        -0.064878459045791162,136.32800000000003,46.642663706148113,136.32800000000003,-0.064874276850442433,
        136.32800000000003,-9.9999999999999982,136.32800000000003,-5.0116575809989987,136.32800000000006,
        -3.355528608733493,136.328,70.0792111192775,68.082011032644715,70.08246539490186,45.319965612648112,
        70.09379964864479,-14.000000000000004,70.093396079164137,-7.0041486765756957,46.64951683334678,
        68.085052658968351,-10.0,68.09450944594461,-5.0077384299939975,68.094221185452341,-3.34867392142978,
        68.094005674607914,46.655237788220333,45.3255467924812,46.675290764014974,-14.0,46.674585386490143,
        -7.0011083270071328,46.6739994865459,-4.6715366480995613,-10.000000000000004,45.342884475415772,
        -5.0044853711592667,45.342358586139262,-3.3429545257648674,45.341962568857838,-9.9999999999999964,
        -13.999999999999998,-9.9999999999999964,0.0047583223517445906,-9.9999999999999982,-6.9916508524709053,
        -9.9999999999999982,0.0047579065103907177,-10.0,-4.6541980426384946,-4.9931510856853736,-14.000000000000004,
        0.0066625962871976127,-14.0,-3.3229015508666389,-14.0,0.0066621668029032488,-14.000000000000004,
        -4.9935534701073809,-6.991938523768094,-4.9938876273720858,-4.65472309775716,-3.3236053682864015,
        -6.9921553113675454,-3.3241928274392922,-4.6551208717229278,140.32799999999997,136.328,140.32799999999997,
        136.32800000000003,140.32799999999997,136.32800000000003,140.32799999999995,68.077963122328043,
        140.32799999999997,-4.68450785771074,140.32799999999997,-13.999999999999998,140.328,-7.0081868651731956,
        70.075282628673619,136.32800000000003,46.642631530347757,136.32800000000003,-0.06488741702733633,136.328,
        -10.000000000000004,136.32800000000006,-5.011674285092937,136.32800000000006,-3.3555583211233451,136.328,
        -3.3555622946665142,136.32800000000006,-9.9999999999999964,136.32800000000003,-10.0,136.328,
        -5.0116580206210077,136.32800000000003,70.093053791180637,-4.6771185392883865,70.093799613272623,
        -14.000000000000002,70.093396046853826,-7.0041488385579989,-10.0,68.094509232290008,-5.0077386181549555,
        68.094221158296435,46.675291532571208,-14.0,46.675291501195034,-14.000000000000004,46.674585433917038,
        -7.0011081945976974,-10.000000000000002,45.342884578934964,-5.0044853494808894,45.342358591863047,
        -9.9999999999999982,-13.999999999999998,-9.9999999999999964,-14.000000000000002,-9.9999999999999982,
        -4.6541960622305716,-9.9999999999999964,-6.9916498557988653,-9.9999999999999964,-6.99164978602478,
        -9.9999999999999947,-4.6541962631244216,-4.9931503007764517,-14.000000000000002,-4.9931493636029334,
        -13.999999999999998,0.0066635162137103814,-14.000000000000002,-4.9935527110051181,-6.9919384142123366,
        -4.9935532626124521,-6.9919374835265442,-3.3236050032142765,-6.9921542921360684,140.32799999999997,136.328,
        140.32799999999997,-13.999999999999998,140.328,-7.0082015385777172,140.32799999999997,-14.000000000000004,
        140.328,-7.0081991580918,140.32799999999997,-13.999999999999998,140.32799999999997,-7.0082004632995671,
        70.0752640337138,136.32800000000006,-5.01167472585953,136.32800000000003,-10.0,136.32800000000003,
        -5.0116769347395431,136.32800000000003,-10.000000000000002,136.328,70.093790333120168,-14.000000000000002,
        -10.000000000000004,68.094499987629192,-9.9999999999999982,68.094509139194315,-10.0,45.342884545523674,
        -9.9999999999999982,-13.999999999999996,-9.9999999999999947,-14.0,-9.9999999999999947,-6.99164961499385,
        -9.9999999999999982,-6.99164878923034,-4.9931489872730346,-13.999999999999996,-3.3228978875299795,-14.0,
        -4.9935525034925687,-6.9919373739570769,140.32799999999997,136.328,140.32799999999997,-13.999999999999998,
        140.328,-14.000000000000002,140.32799999999997,-14.0,-9.9999999999999947,-14.0,-9.9999999999999982,
        -14.000000000000002,140.32799999999997,136.328];
    Explicit_b_F: ARRAY [0..2499] OF LREAL := [-0.12667340248608433,-0.006063437668709459,-8.3619092552944529E-18,
        -0.0061236585018917839,-0.12667628514510906,-5.4210108624275222E-20,-0.031816478047680653,
        -0.0061304672764802117,-0.12667642439759061,-0.0019406208995937544,-0.056510051660952777,
        -0.0061180833246716549,-0.12667579011109506,-0.0031721409299244907,-8.3619092552944529E-18,
        -0.0061236585018917839,-0.12667628514510906,-5.4210108624275222E-20,-0.031816478047680653,
        -0.0061304672764802117,-0.12667642439759061,-0.0019406208995937544,-0.056510051660952777,
        -0.0061180833246716549,-0.12667579011109506,-0.0031721409299244907,-2.9402207665091273E-17,
        -1.7279472123987727E-19,-3.8997820408061615E-17,-0.0061382781607270242,-2.781635022959441E-17,
        -0.001954554803000661,-4.4508616762898093E-17,-0.0061364362134341171,-3.6496532114819666E-17,
        -0.0031976628134779668,-2.9402207665091273E-17,-1.7279472123987727E-19,-2.781635022959441E-17,
        -0.001954554803000661,-3.6496532114819666E-17,-0.0031976628134779668,-0.031817232753816052,
        1.1705995331054431E-18,-0.12667685008982194,-5.6920614055488983E-19,-0.05651137952441581,
        6.1325185381211345E-19,-0.12667674648668509,2.7105054312137611E-19,-7.7886797082401052E-18,
        1.1655173354219173E-18,-0.031817232753816052,1.1705995331054431E-18,-0.05651137952441581,
        6.1325185381211345E-19,-0.031817266661648996,-0.0019560462806767378,-0.03181709911953777,
        -0.0032004303747762012,-0.031817232753816052,-1.8126505071242027E-19,-0.031817266661648996,
        -0.0019560462806767378,-0.056511442169811681,-0.0019531851178935223,-6.2021869980328007E-18,
        -0.001954554803000661,-0.031817266661648996,-0.0019560462806767387,-0.056511442169811681,
        -0.0019531851178935223,-0.056511148498327293,-0.0031951779041220494,-0.056511379524415789,
        -7.555533889508359E-19,-0.056511442169811694,-0.0019531851178935223,-0.056511148498327293,
        -0.0031951779041220494,2.834532230515472E-17,-0.0031976628134779664,-0.031817099119537742,
        -0.0032004303747762012,-0.056511148498327286,-0.0031951779041220485,-2.9402207665091273E-17,
        -1.7279472123987727E-19,-3.8997820408061615E-17,-0.0061382781607270242,-2.781635022959441E-17,
        -0.001954554803000661,-4.4508616762898093E-17,-0.0061364362134341171,-3.6496532114819666E-17,
        -0.0031976628134779668,-0.031817232753816052,1.1705995331054431E-18,-0.12667685008982194,
        -5.6920614055488983E-19,-0.05651137952441581,6.1325185381211345E-19,-0.12667674648668509,
        2.7105054312137611E-19,-0.031817266661648996,-0.0019560462806767378,-0.03181709911953777,
        -0.0032004303747762012,-0.056511442169811681,-0.0019531851178935223,-0.056511148498327293,
        -0.0031951779041220494,-3.1637633492013779E-17,-2.1218175328720223E-19,-2.9586609384686495E-17,
        -1.2874900798265365E-18,-3.629303244924182E-17,-1.3844753522871539E-18,-3.5260975742571659E-17,
        -0.0019546071360561261,-3.7007716498487636E-17,-0.0032030047769573962,-2.9586609384686495E-17,
        -1.2874900798265365E-18,-3.5260975742571659E-17,-0.0019546071360561261,-0.031819629222642885,
        -5.5904174518783822E-20,-0.056511639234444355,6.7762635780344027E-19,-0.12667689109875555,
        4.87890977618477E-19,1.3640969307162975E-17,4.0657581468206416E-20,-0.031817379490146271,
        2.6427427954334171E-19,-0.056511639234444355,6.7762635780344027E-19,-0.0565116579667842,
        -1.2197274440461925E-19,-9.9828126789839634E-18,-2.1747570920754161E-19,-1.4679504492390652E-17,
        -4.4045713257223618E-20,-0.031819629222642885,-5.5904174518783822E-20,-0.031819495581118705,
        -0.0032010631169945782,-0.031817379490146284,2.6935647722686751E-19,-0.031817277135142374,
        -0.0019560987878057871,-9.8746042199722266E-18,-0.0019574634784031352,-0.031819663167738495,
        -0.0019563921511248318,-0.056511639234444369,-6.6068569885835426E-19,-0.056511591038165096,
        -3.3203691532368573E-19,-0.056511460878431695,-0.0019532373498035932,6.2570323813675166E-18,
        -0.0032030047769573944,-0.031819495581118684,-0.003201063116994579,-3.629303244924182E-17,
        -1.3844753522871539E-18,-5.39196557327058E-17,-1.3755815063409838E-18,-2.2981062650193236E-17,
        -0.0032037800282279736,-3.1515396049813143E-17,-0.0019574634784031361,-3.5260975742571659E-17,
        -0.0019546071360561261,-3.7007716498487636E-17,-0.0032030047769573962,-0.031819629222642885,
        -5.5904174518783822E-20,-0.031817351949048972,2.2700482986415249E-19,-0.12667689109875555,
        4.87890977618477E-19,-0.031819663167738495,-0.0019563921511248322,-0.031817277135142374,
        -0.0019560987878057871,-0.056511460878431688,-0.0019532373498035924,-4.5264312426914288E-17,
        -6.4374503991326826E-20,-1.8829860054818317E-17,-1.4162771898161559E-18,-9.05149995347786E-18,
        -0.0019582276830549272,-4.01097761444595E-17,-1.7999450129153882E-20,-3.2785416075102559E-17,
        -0.0019575161121738087,-4.5264312426914288E-17,-6.4374503991326826E-20,-8.1940908526196947E-18,
        -0.0019579342315898221,-0.031819776023428871,-6.9287295085401768E-19,-0.031819776023428878,
        -6.8609668727598327E-19,-2.6619971612698751E-17,3.5575383784680614E-19,-0.031819786518259209,
        8.7752613335545515E-19,-1.8776920495614923E-17,-1.4095957935146237E-18,-0.031819748476883458,
        -1.1892342579450377E-18,-1.1073949933725112E-17,-0.0019575161121738074,1.2611473551669278E-17,
        -0.0019582276830549259,7.93648695753598E-18,-0.0032044132383236136,-3.4094373146186072E-17,
        -1.3349239248727773E-18,-4.5264312426914288E-17,-6.4374503991326826E-20,-9.0567409698389962E-18,
        -0.001958227683054928,-5.43860797190673E-17,-0.0019575161121738087,-0.031817389976958411,
        -1.5280474368467578E-18,-0.0565116579667842,-1.2197274440461925E-19,-0.031819673649245137,
        -0.0019564446946577791,-4.0445883408782404E-17,-2.0629487430378485E-18,-1.4750814078637623E-17,
        -8.2818133307315491E-19,-4.0447185391066563E-17,6.3866284222974246E-19,-4.8277910069457279E-17,
        -9.9229909770841285E-19,-2.6619429395807223E-17,-9.9568722949743E-19,-4.0445883408782404E-17,
        -2.0629487430378485E-18,-4.3236735011029394E-17,-1.334067109051033E-18,-0.010939895258464375,
        -0.12940337663776541,1.8973538018496328E-19,-0.12940857748967641,-0.011001415774033131,
        -1.1907589172500954E-17,-0.0034622111951241163,-0.12940866066139117,-0.011010925708052186,
        -0.032495995972325727,-0.005684687311205988,-0.12940746957634541,-0.010999089451642668,-0.0577221130716327,
        1.8973538018496328E-19,-0.12940857748967641,-0.011001415774033131,-1.1907589172500954E-17,
        -0.0034622111951241163,-0.12940866066139117,-0.011010925708052186,-0.032495995972325727,
        -0.0056846873112059888,-0.12940746957634541,-0.010999089451642668,-0.057722113071632712,
        -1.8499199568033919E-18,-3.1316290367649179E-17,-2.5207700510287978E-18,-0.12940951062758926,
        -3.3627208005995723E-18,-0.032497207130407976,-2.3445871979999033E-18,-0.12940931580424303,
        -1.5958100726271018E-18,-0.057724329102651205,-1.8499199568033919E-18,-3.1316290367649179E-17,
        -3.3627208005995723E-18,-0.032497207130407976,-1.5856456772600502E-18,-0.057724329102651212,
        -0.0034781423641150754,-1.4472616695023789E-17,-0.011018053990055782,-1.9238659330986924E-17,
        -0.0057127737954156535,4.3457025358881879E-18,-0.011016492215632667,-1.3649088912055796E-17,
        -5.1838416371963181E-19,1.1910130271342717E-17,-0.0034781423641150754,-1.4472616695023789E-17,
        -0.0057127737954156543,4.3465495688354422E-18,-0.0034805192947300781,-0.032497220518183073,
        -0.0034774059198201877,-0.057724356242492864,-0.0034781423641150754,7.140911261827379E-18,
        -0.0034805192947300781,-0.032497220518183073,-0.00571704223028016,-0.032496943931058939,
        -6.7593229190893167E-19,-0.032497207130407955,-0.0034805192947300781,-0.032497220518183059,
        -0.0057170422302801607,-0.032496943931058939,-0.0057115870095412712,-0.057723849103550343,
        -0.0057127737954156535,4.3457025358881879E-18,-0.0057170422302801616,-0.032496943931058932,
        -0.0057115870095412712,-0.05772384910355035,3.7980957354882827E-18,-0.057724329102651191,
        -0.0034774059198201864,-0.057724356242492864,-0.00571158700954127,-0.057723849103550329,
        -1.8499199568033919E-18,-3.1316290367649179E-17,-2.5207700510287978E-18,-0.12940951062758926,
        -3.3627208005995723E-18,-0.032497207130407976,-2.3445871979999033E-18,-0.12940931580424303,
        -1.5856456772600502E-18,-0.057724329102651212,-0.0034781423641150754,-1.4472616695023789E-17,
        -0.011018053990055782,-1.9238659330986924E-17,-0.0057127737954156543,4.3465495688354422E-18,
        -0.011016492215632667,7.9917558573443237E-18,-0.0034805192947300781,-0.032497220518183073,
        -0.0034774059198201877,-0.057724356242492864,-0.0057170422302801607,-0.032496943931058939,
        -0.005711587009541272,-0.05772384910355035,-1.1180834903756764E-18,-2.8703842234969904E-17,
        -2.2514135738019303E-18,-1.6261338521388058E-17,-2.1785687403380605E-18,-3.0005983337805979E-17,
        -2.4496192834594366E-18,-0.032499690181368147,-2.4530074152484538E-18,-0.057724640166312291,
        -2.2514135738019303E-18,-1.6261338521388058E-17,-2.447925217564928E-18,-0.032499690181368147,
        -0.0034782384082034431,-2.9130521847259457E-18,-0.0057203209764982678,-1.5056010637445189E-17,
        -0.011020049672395411,1.9245435594564958E-17,1.7885100681274552E-18,5.3299548205976849E-18,
        -0.0034823937966747143,-4.7944182396961535E-18,-0.0057203209764982686,-1.5054740088024307E-17,
        -0.0057212109064913585,-3.6574882662440689E-17,2.1345230270808369E-19,1.4522843101818009E-17,
        -8.3348042009823153E-19,-8.3925083205140145E-18,-0.0034782384082034418,-2.9136874594363864E-18,
        -0.0034775019361867527,-0.057724381593873116,-0.0034823937966747156,1.6840391419954779E-17,
        -0.003481014589598143,-0.032499703597191981,3.1001405869507392E-19,-0.03249737675610765,
        -0.0034806155086637754,-0.032497234404046518,-0.0057203209764982695,-1.499333019934837E-17,
        -0.0057195819017150417,7.3615633445871242E-18,-0.0057179316027686257,-0.032499426937493366,
        2.9341221292888964E-18,-0.057724640166312263,-0.0034775019361867514,-0.057724381593873109,
        -2.1751806085490433E-18,-3.0005401002654742E-17,-2.1590869825512116E-18,-1.8180291663392675E-17,
        -2.6393546636444E-18,-0.057724722338242183,-1.0333801956502464E-18,-0.032497376756107664,
        -2.447925217564928E-18,-0.032499690181368147,-2.4496192834594366E-18,-0.057724640166312291,
        -0.0034782384082034418,-2.9136874594363864E-18,-0.0034819660630087974,-1.42590585131973E-17,
        -0.011020049672395411,-2.3488223627361748E-18,-0.0034806155086637754,-0.032497234404046539,
        -0.003481014589598143,-0.032499703597191981,-0.0057179316027686248,-0.032499426937493379,
        -2.4321715627988556E-19,-2.4769572718320691E-17,-3.2932640989247197E-18,-4.3098028973033865E-17,
        -3.0493186101154812E-20,-0.032497435184955785,-1.1608586542120186E-18,-7.0482140936622365E-18,
        -1.7508171019746388E-18,-0.032499859870392257,-2.3045448321122832E-19,-4.6363830675621824E-17,
        -1.2468324983583301E-18,-0.032499904406537286,-0.0034824901317153855,-1.3784825941853297E-17,
        -0.0034824901317153868,-3.5417518019136094E-17,2.2535452699392677E-19,-1.0840645296315756E-17,
        -0.0034829857776749878,-6.0625324408542479E-18,-5.8614679949997583E-19,-4.309872711347086E-17,
        -0.0034820623747332268,-5.69567188348657E-17,9.4867690092481638E-19,-0.032499859870392236,
        2.6495190590114515E-18,-0.032497435184955743,2.8426425709854319E-18,-0.05772474772329142,
        -1.74022919013396E-18,-3.8454607591075591E-17,-2.3045448321122832E-19,-4.6363830675621824E-17,
        -4.072534410398676E-18,-0.0324974351849558,-3.0823528950583989E-18,-0.032499859870392278,
        -0.0034828894057362539,-1.4940390640144977E-17,-0.0057212109064913577,-1.4962837013247215E-17,
        -0.0034811108404072628,-0.032499717489793044,-4.6570117914014579E-19,-5.4131969834891012E-17,
        -7.75458663211312E-19,-5.4659205244755268E-17,-4.7875783090603467E-19,-1.0848096539273634E-17,
        -1.1109398035093036E-18,-5.4060977885999261E-17,-2.4568260686969107E-18,-5.4074900990069754E-17,
        8.7612459859210622E-19,-3.2500058616106466E-17,-2.7055760048624738E-18,-2.1687985305904772E-17,
        -0.021835439137868347,-0.0011520122606157824,8.3760970571609625E-19,-0.0011623928796879576,
        -0.021835986823640203,2.9815559743351372E-19,-0.0046660193730712375,-0.0011641448432321742,
        -0.021836028047420925,-0.00034855849507587592,-0.0088399634659200779,-0.0011621335886920921,
        -0.021835908054478017,-0.00058417725377516751,8.3760970571609625E-19,-0.0011623928796879576,
        -0.021835986823640203,2.9815559743351372E-19,-0.0046660193730712375,-0.0011641448432321742,
        -0.021836028047420925,-0.00034855849507587592,-0.0088399634659200761,-0.0011621335886920921,
        -0.021835908054478017,-0.00058417725377516751,-1.1794933790516132E-19,3.5151867311053464E-19,
        -1.6721489169983957E-18,-0.0011652903420256554,-2.9172079401234121E-18,-0.00035096037140803615,
        -2.1520989607363636E-18,-0.0011650045622868016,-2.9730327053033908E-18,-0.00058857662244823472,
        -1.1794933790516132E-19,3.5151867311053464E-19,-2.9172079401234121E-18,-0.00035096037140803615,
        -2.9730327053033908E-18,-0.00058857662244823472,-0.0046661626879632477,3.7269449679189215E-19,
        -0.021836104506786864,2.2869889575866109E-19,-0.0088402156943794986,4.7137383514701814E-19,
        -0.021836084179334414,3.1340219048409113E-19,-2.8197197418503624E-18,3.5278922253141609E-19,
        -0.0046661626879632477,3.7269449679189215E-19,-0.0088402156943794968,4.6925625277888239E-19,
        -0.0046661729227340945,-0.00035135054557220417,-0.00466614122182821,-0.00058929774581286808,
        -0.0046661626879632477,3.7269449679189215E-19,-0.0046661729227340945,-0.00035135054557220417,
        -0.0088402343122757146,-0.00035088561017350455,-2.1543753617821095E-19,-0.00035096037140803615,
        -0.0046661729227340919,-0.000351350545572204,-0.0088402343122757129,-0.00035088561017350455,
        -0.0088401787462571157,-0.00058844410776131336,-0.0088402156943794986,3.0239076216978522E-19,
        -0.00884023431227572,-0.00035088561017350455,-0.0088401787462571157,-0.00058844410776131336,
        2.430455163027808E-18,-0.00058857662244823472,-0.0046661412218282064,-0.00058929774581286819,
        -0.00884017874625711,-0.00058844410776131336,-1.1794933790516132E-19,3.5151867311053464E-19,
        -1.6721489169983957E-18,-0.0011652903420256554,-2.9172079401234121E-18,-0.00035096037140803615,
        5.4284224007159973E-19,-0.0011650045622868016,-2.9730327053033908E-18,-0.00058857662244823472,
        -0.0046661626879632477,3.7269449679189215E-19,-0.021836104506786864,2.2869889575866109E-19,
        -0.0088402156943794968,4.6925625277888239E-19,-0.021836084179334414,3.1340219048409113E-19,
        -0.0046661729227340945,-0.00035135054557220417,-0.00466614122182821,-0.00058929774581286808,
        -0.0088402343122757129,-0.00035088561017350455,-0.0088401787462571123,-0.00058844410776131336,
        -1.3346592270767604E-18,2.82326669231699E-19,-1.99168547890518E-19,2.2658131339052534E-19,
        -1.578684125224804E-18,2.3727510434961088E-19,-8.3673620298924025E-19,-0.00035097205163314076,
        3.0059081715686983E-19,-0.00058966848483959448,-1.99168547890518E-19,2.2658131339052534E-19,
        -8.3673620298924025E-19,-0.00035097205163314076,-0.004666697129121284,4.8174998875088332E-19,
        -0.008840269714523688,4.3410438546782892E-19,-0.021836113712710516,2.0837010502455788E-19,
        7.9059491036817479E-18,3.9048218868423246E-19,-0.0046661931893067525,4.5655075857006788E-19,
        -0.0088402697145236846,4.3198680309969317E-19,-0.0088402739021540347,5.6158284402960112E-19,
        1.3670317675296357E-18,4.4993331366964366E-19,-1.5821516663526262E-18,4.0562290261640307E-19,
        -0.0046666971291212866,4.8302053817176477E-19,-0.0046666756618988928,-0.00058943885502096274,
        -0.0046661931893067577,2.9116757561866574E-19,-0.0046661752611696682,-0.00035136226893268138,
        -1.4712035851521137E-18,-0.0003515548854198116,-0.004666707372365379,-0.00035142767883477574,
        -0.008840269714523688,9.6561755986990239E-20,-0.0088402602471837673,2.9730856448625942E-19,
        -0.0088402384954132315,-0.00035089728892171812,3.0045846825886135E-19,-0.00058966848483959437,
        -0.0046666756618988928,-0.00058943885502096285,-1.5888485205918556E-18,2.3611043404713622E-19,
        -6.3560558268574647E-19,3.1890790464124408E-19,-1.3013867141174274E-18,-0.00058978898971890226,
        -1.4744726029329233E-18,-0.00035155488541981176,-8.3673620298924025E-19,-0.00035097205163314076,
        2.9381455357883543E-19,-0.00058966848483959448,-0.0046666971291212866,4.8302053817176477E-19,
        -0.004666187775523677,4.7222086809427244E-19,-0.021836113712710516,2.0837010502455788E-19,
        -0.0046667073723653842,-0.00035142767883477574,-0.0046661752611696682,-0.00035136226893268138,
        -0.0088402384954132263,-0.00035089728892171796,-1.8489761437244689E-18,1.232432938255007E-19,
        -1.4251329337553603E-19,1.5386230185264307E-19,-2.7136156303169605E-18,-0.00035169687999964154,
        -4.9415935230040384E-19,4.258458142320995E-19,5.2317519382753894E-19,-0.00035156662712727745,
        -1.8489761437244689E-18,1.232432938255007E-19,-2.4459399840948007E-19,-0.00035163144666093126,
        -0.0046667276446882341,4.1102273765514924E-19,-0.0046667276446882315,4.0890515528701349E-19,
        -9.5356553834500477E-19,4.2679872629776058E-19,-0.00466672998743669,5.14784273693801E-19,
        -1.4592789494415493E-19,3.2237967214500863E-19,-0.0046667222297373193,1.0630263488041469E-19,
        5.2647068138795021E-19,-0.00035156662712727729,2.6900972311408528E-18,-0.00035169687999964138,
        -5.7968817327716179E-20,-0.00058993018680938666,1.5512217288880434E-18,2.3791037906005161E-19,
        -1.8489761437244689E-18,1.232432938255007E-19,-1.6953893834886855E-20,-0.00035169687999964171,
        -4.890516774540114E-18,-0.00035156662712727745,-0.0046661955302668917,3.2441361879839703E-19,
        -0.0088402739021540312,5.5946526166146537E-19,-0.00466670971258821,-0.00035143941031378837,
        -2.460318683737051E-18,2.4156320864508578E-19,-1.9600474748362518E-18,2.4520144624712663E-19,
        -2.4653401353443424E-18,2.413514504082722E-19,-9.535282635186516E-19,2.5770977420212088E-19,
        -9.47597120032705E-19,2.5845092803096839E-19,-2.460318683737051E-18,2.4156320864508578E-19,
        -2.7015815614391379E-18,1.7057475020245581E-19,-0.0034982247754591846,-0.037913871321265488,
        3.2864878353466853E-19,-0.03791553438554341,-0.003516249659905755,6.0562855728682474E-20,
        -0.0010483412940467669,-0.037915602504622059,-0.00352001142228519,-0.0081901839499625134,
        -0.0017637665131279233,-0.037915222177636647,-0.003516769828667967,-0.015456721801501918,
        3.2864878353466853E-19,-0.03791553438554341,-0.003516249659905755,6.0562855728682474E-20,
        -0.0010483412940467669,-0.037915602504622059,-0.00352001142228519,-0.0081901839499625134,
        -0.0017637665131279229,-0.037915222177636647,-0.003516769828667967,-0.015456721801501924,
        -2.0159384144652348E-19,-1.1845226371759356E-18,-4.7433845046240819E-20,-0.037915859870396064,
        -9.1564261598189867E-19,-0.0081905711372341986,-4.8111471404044259E-19,-0.037915794999810175,
        -3.7438856268640075E-19,-0.015457430339336756,-2.0159384144652348E-19,-1.1845226371759356E-18,
        -9.1564261598189867E-19,-0.0081905711372341986,-3.6930636500287495E-19,-0.015457430339336761,
        -0.0010530089868256581,5.6347808024908262E-18,-0.0035218080110374283,-2.732951804316E-18,
        -0.0017719955998451308,3.356897449087199E-18,-0.0035214299089605374,8.1734444245303711E-18,
        -2.0413494028828638E-19,4.2188593520368564E-18,-0.0010530089868256581,5.6347808024908262E-18,
        -0.0017719955998451308,3.356897449087199E-18,-0.0010539568187064221,-0.0081905849637701356,
        -0.0010531016854318472,-0.015457456534433,-0.0010530089868256581,5.6347808024908262E-18,
        -0.0010539568187064221,-0.0081905849637701356,-0.0017736905237788257,-0.0081904966580441437,
        4.3113977015243887E-19,-0.0081905711372341934,-0.0010539568187064217,-0.00819058496377013,
        -0.0017736905237788255,-0.0081904966580441437,-0.0017721939819592,-0.015457294593549919,
        -0.0017719955998451308,-2.0464316005663896E-18,-0.0017736905237788266,-0.0081904966580441437,
        -0.0017721939819592,-0.015457294593549924,9.7493492228969969E-19,-0.015457430339336754,
        -0.0010531016854318466,-0.015457456534433001,-0.0017721939819591993,-0.015457294593549914,
        -2.0159384144652348E-19,-1.1845226371759356E-18,-4.7433845046240819E-20,-0.037915859870396064,
        -9.1564261598189867E-19,-0.0081905711372341986,-4.8450284582945979E-19,-0.037915794999810175,
        -3.6930636500287495E-19,-0.015457430339336761,-0.0010530089868256581,5.6347808024908262E-18,
        -0.0035218080110374283,-2.732951804316E-18,-0.0017719955998451308,3.356897449087199E-18,
        -0.0035214299089605374,8.18699695168644E-18,-0.0010539568187064221,-0.0081905849637701356,
        -0.0010531016854318472,-0.015457456534433004,-0.0017736905237788255,-0.0081904966580441437,
        -0.0017721939819591997,-0.015457294593549924,-4.7010328572613669E-19,-1.3141914699997482E-19,
        -8.4385657370209671E-20,-1.1857402470376137E-18,-8.6736173798840355E-19,-3.407203265220224E-18,
        -5.8720559068404371E-19,-0.0081914952946237352,-2.388632911257127E-19,-0.015457540044886605,
        -8.4385657370209671E-20,-1.1857402470376137E-18,-5.9038196423624734E-19,-0.0081914952946237282,
        -0.001053044746302335,1.5328649367342666E-18,-0.0017745168956370212,2.7445985073407467E-18,
        -0.0035225506987666363,7.3653749928497686E-18,1.262820245237755E-18,9.6305528520445813E-18,
        -0.0010544292673404124,7.4725246606774376E-18,-0.001774516895637021,2.7442808699855263E-18,
        -0.0017748480792266457,-1.0456621733854338E-18,-4.70950318673391E-19,5.2720720300536742E-18,
        -1.9566461081574338E-19,1.9956890330699367E-18,-0.0010530447463023354,1.5330766949710802E-18,
        -0.0010531374576252502,-0.015457465979431909,-0.0010544292673404132,2.0594017925712211E-18,
        -0.001054141160788231,-0.0081915091323479083,3.2314306937751558E-19,-0.00819063094036294,
        -0.0010539926448452485,-0.0081905901342984883,-0.0017745168956370219,-8.0768826685433809E-18,
        -0.001774334854501361,-4.3972656665522934E-18,-0.001774021536753176,-0.0081914208010279415,
        4.2775163836342167E-19,-0.015457540044886595,-0.0010531374576252493,-0.015457465979431904,
        -8.6820877093565785E-19,-3.4073620838978341E-18,-3.4050724479622874E-19,-2.993361496037494E-18,
        -2.447925217564928E-19,-0.015457567403298908,-3.4813054132151744E-19,-0.0081906309403629463,
        -5.9038196423624734E-19,-0.0081914952946237282,-2.405573570202213E-19,-0.015457540044886605,
        -0.0010530447463023354,1.5330766949710802E-18,-0.0010543228028200187,5.2656332561655615E-18,
        -0.0035225506987666363,7.3810451023739732E-18,-0.0010539926448452492,-0.0081905901342984935,
        -0.001054141160788231,-0.0081915091323479083,-0.0017740215367531753,-0.0081914208010279415,
        -4.6609629359195911E-19,-4.648622693650007E-19,-2.7782680669941051E-19,3.4962161709370553E-18,
        -1.7575933655526732E-19,-0.00819065093434982,-3.6348301349050163E-19,1.1533177448757402E-17,
        8.9573734172142261E-20,-0.00819155512097787,-4.6485265339037978E-19,-4.55227269589983E-19,
        -6.9393174203808555E-19,-0.0081915699426062215,-0.0010544651240993646,-2.1534753892756518E-18,
        -0.0010544651240993646,-2.1535812683940586E-18,-1.4930700529461648E-20,-2.1646721060471696E-18,
        -0.0010546495763118805,4.4861511864547916E-18,4.0064658405128406E-19,-1.907404046292152E-18,
        -0.0010543586543143618,-2.3973149989664835E-18,8.1950437646853558E-20,-0.00819155512097786,
        4.921261423547485E-19,-0.0081906509343498083,3.5998900258307764E-19,-0.015457576859199004,
        -4.6120943977996653E-19,1.749573022333359E-18,-4.6485265339037978E-19,-4.55227269589983E-19,
        -8.4745646372792749E-19,-0.0081906509343498256,8.8726701224887961E-20,-0.00819155512097787,
        -0.001054613705821476,-5.1583777092194857E-18,-0.0017748480792266462,-1.0256510200065509E-18,
        -0.0010541770006516429,-0.0081915143053841559,4.1312398320618707E-20,-3.1012490089715603E-18,
        -1.0894961284058438E-18,5.3833863454703946E-18,4.23171206500766E-20,7.7514036411160156E-18,
        -1.3193265813930833E-20,-2.1547194689169316E-18,-1.1759897521695683E-20,-7.5663467944756522E-18,
        4.5249235199094131E-20,-8.4940530125110242E-18,5.4294849001241571E-22,-5.4233692790932017E-18,
        -0.90852126123084109,-0.043908146081154252,1.1237416704633352E-16,-0.044340059223466725,
        -0.90854213589311628,5.4210108624275222E-18,-0.22499743169378195,-0.044391150716473024,-0.90854320277576739,
        -0.013973130057841329,-0.40175302414947389,-0.044302834795567785,-0.90853861186181406,-0.02289738328452481,
        1.1237416704633352E-16,-0.044340059223466725,-0.90854213589311628,5.4210108624275222E-18,
        -0.22499743169378195,-0.044391150716473024,-0.90854320277576739,-0.013973130057841329,-0.40175302414947389,
        -0.044302834795567785,-0.90853861186181406,-0.02289738328452481,-2.0211137857729586E-16,
        -3.3610267347050637E-18,1.4233541645661263E-17,-0.044446387153773116,-1.2255042087464668E-16,
        -0.014073066200566241,-1.7068052700353054E-16,-0.044433312973263257,-1.4178653910679184E-16,
        -0.02308043023166,-2.0211137857729586E-16,-3.3610267347050637E-18,-1.2254660922638404E-16,
        -0.014073066200566246,-1.4178653910679184E-16,-0.02308043023166,-0.22500289657472694,1.6127507315721878E-18,
        -0.90854626790451765,5.4210108624275222E-19,-0.4017626395980568,1.0543866127421531E-17,-0.90854551524313676,
        7.48099499014998E-18,-2.9203154922486513E-17,7.37257477290143E-18,-0.22500289657472694,
        1.6127507315721878E-18,-0.40176263959805669,1.0489656018797255E-17,-0.2250031571391346,
        -0.014084282907403574,-0.22500194445913865,-0.023101232532859166,-0.22500289657472694,
        1.7821573210230479E-17,-0.2250031571391346,-0.014084282907403586,-0.40176311984350016,-0.014063877541696803,
        -1.2255465603938295E-16,-0.014073066200566236,-0.2250031571391346,-0.014084282907403574,
        -0.40176311984350005,-0.014063877541696803,-0.4017609942320583,-0.023063772260979193,-0.40176263959805669,
        5.0957502106818708E-18,-0.40176311984350022,-0.014063877541696813,-0.4017609942320583,-0.023063772260979193,
        2.0403837853229939E-16,-0.02308043023166,-0.22500194445913849,-0.023101232532859169,-0.401760994232058,
        -0.023063772260979186,-2.0211137857729586E-16,-3.3610267347050637E-18,1.4233541645661263E-17,
        -0.044446387153773116,-1.2254660922638404E-16,-0.014073066200566246,1.9888333601530972E-18,
        -0.044433312973263257,-1.4178653910679184E-16,-0.02308043023166,-0.22500289657472694,1.6127507315721878E-18,
        -0.90854626790451765,5.9631119486702744E-18,-0.40176263959805669,1.0489656018797255E-17,
        -0.90854551524313676,7.48099499014998E-18,-0.2250031571391346,-0.014084282907403586,-0.22500194445913865,
        -0.023101232532859166,-0.40176311984350005,-0.014063877541696808,-0.40176099423205819,-0.023063772260979193,
        -1.1948500863853337E-16,-7.8316666303132609E-18,-1.0077230382823216E-16,-2.5478751053409354E-18,
        -4.0905762121751926E-17,1.6703489719854803E-18,-8.65074749030817E-18,-0.014073452133259199,
        -5.3407121390278145E-17,-0.023119416718676764,-1.0077092739969287E-16,-2.5343225781848666E-18,
        -8.643971226730135E-18,-0.014073452133259209,-0.22502056771591866,8.2263839837337649E-18,
        -0.40176453880416918,6.5323180892251642E-18,-0.90854657053851451,5.5294310796760726E-18,
        2.45051555019675E-16,2.6834003769016235E-18,-0.22500396954755839,9.4867690092481638E-19,
        -0.40176453880416907,6.478107980600889E-18,-0.40176467697335466,-2.439454888092385E-19,
        5.3732382042023796E-17,8.3331101350878067E-18,-4.1341984089587891E-17,7.0235971986326584E-18,
        -0.22502056771591855,8.1518450843753865E-18,-0.22501961554900995,-0.023105898263657981,-0.22500396954755847,
        1.1858461261560205E-17,-0.225003234379625,-0.014084670139843564,-5.3978445113201171E-17,
        -0.014094294168846267,-0.22502082855573682,-0.014086833295573026,-0.40176453880416929,
        6.6407383064737147E-18,-0.40176418862008356,6.3967928176644762E-18,-0.40176325784096573,
        -0.014064262811759857,1.1939607017907167E-16,-0.023119416718676764,-0.22501961554900987,
        -0.023105898263657981,-4.1339442990746128E-17,1.6195269951502222E-18,-4.3272795692854069E-18,
        2.1819568721270777E-18,-8.3520836731063031E-17,-0.023124920378727248,-5.4079242033924432E-17,
        -0.014094294168846278,-8.643971226730135E-18,-0.014073452133259209,-2.2653726767726812E-16,
        -0.023119416718676764,-0.22502056771591855,8.1518450843753865E-18,-0.22500376942411082,
        4.2283884726934673E-18,-0.90854657053851451,1.0950441942103595E-17,-0.225020828555737,-0.014086833295573026,
        -0.225003234379625,-0.014084670139843564,-0.4017632578409655,-0.014064262811759858,-6.8140584528386856E-17,
        -4.7298319774680131E-18,-1.5717712775840248E-16,-4.8427867988345792E-18,-1.8241786255363338E-16,
        -0.014099813725742058,-9.7153620258884181E-18,1.44774871344705E-17,-1.9124479289697044E-16,
        -0.014094682296279696,-6.8139128690508763E-17,-4.7162794503119443E-18,-6.6146920433456449E-17,
        -0.014097649905087963,-0.22502164116342194,6.8711312681268844E-18,-0.2250216411634221,
        1.5517643593698782E-18,-1.0201159574812646E-16,2.2158381900172497E-18,-0.22502171855946634,
        2.1480755542369057E-18,1.5798011499239956E-17,4.91865166871488E-19,-0.22502144099999252,
        2.6766241133235891E-18,-1.8120999357084874E-17,-0.014094682296279686,-9.6193296654934618E-18,
        -0.014099813725742047,1.9217822320484468E-16,-0.023129589494450122,-1.5185585502551415E-16,
        -3.1611269591530489E-18,-6.8139128690508763E-17,-4.7162794503119443E-18,-9.698950762535366E-18,
        -0.014099813725742063,-1.9135406014716624E-16,-0.014094682296279696,-0.22500404688447739,
        8.40256683676266E-18,-0.40176467697335472,1.0625181290357943E-17,-0.22502090585531667,-0.0140872207964491,
        -2.8013481348918148E-16,5.2482161411876449E-18,-1.0580415599095554E-16,-2.786738913454531E-18,
        -1.0705883760614638E-16,1.0608240631412857E-17,-1.0176638301861879E-16,2.2463313761184045E-18,
        -1.0165657313794115E-16,-3.1509625637859973E-18,-2.8013342961601668E-16,5.2583805365546965E-18,
        -5.7474348667278365E-20,-2.9607205860406696E-20,-0.077953938048960669,-0.91495630205656719,
        1.5395670849294163E-17,-0.91499336154188149,-0.078388923478923359,-1.2000762796698927E-17,
        -0.024548090137893282,-0.91499404071464974,-0.0784581439271197,-0.22706440144138565,-0.040393877243513461,
        -0.91498555513722191,-0.07837495020825766,-0.405131234178429,1.5395670849294163E-17,-0.91499336154188149,
        -0.078388923478923359,-1.2000762796698927E-17,-0.024548090137893282,-0.91499404071464974,
        -0.0784581439271197,-0.22706440144138565,-0.040393877243513461,-0.91498555513722191,-0.07837495020825766,
        -0.405131234178429,-1.2197274440461925E-18,-6.8118389618190833E-17,-4.9873299934333204E-18,
        -0.91500006722362592,-4.8382521947165635E-18,-0.22707303152550876,-3.2526065174565133E-18,
        -0.91499867394199985,-9.7849246066816775E-18,-0.4051470246964986,-1.2197274440461925E-18,
        -6.8118389618190833E-17,-4.8382521947165635E-18,-0.22707303152550876,-9.7849246066816775E-18,
        -0.4051470246964986,-0.024660732712307117,1.417594340524797E-17,-0.078507952497007219,
        1.9447876468958736E-17,-0.040592464909515784,1.8488357546309064E-16,-0.078497094095205028,
        7.5948362182609586E-17,-1.3823577699190182E-18,2.7769805769142786E-16,-0.024660732712307103,
        1.4168320108722682E-17,-0.040592464909515784,1.8488357546309064E-16,-0.024678049245177087,
        -0.22707314681162666,-0.02465616095779212,-0.405147254584257,-0.024660732712307117,1.8708416706005732E-16,
        -0.024678049245177087,-0.22707314681162666,-0.0406235469714099,-0.22707117636130061,5.9089018400459992E-18,
        -0.22707303152550867,-0.024678049245177074,-0.22707314681162657,-0.0406235469714099,-0.22707117636130061,
        -0.040585198407018679,-0.405143641589301,-0.040592464909515784,1.1975351808281298E-17,-0.040623546971409907,
        -0.2270711763613007,-0.040585198407018679,-0.405143641589301,1.1763593571467723E-17,-0.40514702469649849,
        -0.0246561609577921,-0.405147254584257,-0.040585198407018672,-0.405143641589301,-1.2197274440461925E-18,
        -6.8118389618190833E-17,-4.9873299934333204E-18,-0.91500006722362592,-4.8382521947165635E-18,
        -0.22707303152550876,-3.2526065174565133E-18,-0.91499867394199985,-9.7849246066816775E-18,
        -0.4051470246964986,-0.024660732712307103,1.4168320108722682E-17,-0.078507952497007219,
        1.9447876468958736E-17,-0.040592464909515784,1.8488357546309064E-16,-0.078497094095205028,
        7.5948362182609586E-17,-0.024678049245177087,-0.22707314681162666,-0.024656160957792109,-0.405147254584257,
        -0.0406235469714099,-0.22707117636130061,-0.040585198407018679,-0.405143641589301,-1.4094628242311558E-18,
        6.5815518792843204E-18,-1.4894227344519617E-17,-4.6953577365147631E-17,7.3183646642771549E-19,
        -1.4633468251707381E-16,5.2922618544448685E-18,-0.22709100233229687,-9.5680841721845766E-18,
        -0.40514926269585039,-1.4894227344519617E-17,-4.6953577365147631E-17,5.2922618544448685E-18,
        -0.22709100233229687,-0.02466142784965503,1.1036924006018259E-16,-0.040646457087583146,
        1.5888644024596166E-17,-0.0785223958657716,8.3937576941112146E-17,2.8192644616412132E-17,
        2.9900517147960978E-16,-0.02469114725936063,9.6381337969225073E-17,-0.040646457087583146,
        1.5888644024596166E-17,-0.040652897782438434,1.9426361832098477E-16,-1.5178830414797062E-18,
        1.7948585800671261E-16,6.5052130349130266E-19,2.657311762126191E-17,-0.02466142784965503,
        1.1037008709312984E-16,-0.024656855942051376,-0.40514743808224646,-0.024691147259360651,
        9.639658456227565E-17,-0.024681633887332338,-0.22709111782296573,7.15573433840433E-18,-0.22707425188322058,
        -0.024678745617735788,-0.22707324731405812,-0.040646457087583153,1.5893726222279692E-17,
        -0.040641311777483369,4.953956895311501E-17,-0.04062998370810441,-0.22708914685042259,
        1.0299920638612292E-18,-0.40514926269585017,-0.024656855942051355,-0.40514743808224646,
        7.3183646642771549E-19,-1.4633468251707381E-16,-2.0464316005663896E-18,-2.880081427254072E-17,
        6.2341624917916505E-18,-0.40514985034555978,7.26415455565288E-18,-0.22707425188322075,
        5.2922618544448685E-18,-0.22709100233229687,-9.5680841721845766E-18,-0.40514926269585039,
        -0.02466142784965503,1.1037008709312984E-16,-0.02468816702271235,1.2348385118252092E-16,-0.0785223958657716,
        8.3937576941112146E-17,-0.0246787456177358,-0.22707324731405804,-0.024681633887332327,-0.22709111782296573,
        -0.040629983708104396,-0.22708914685042267,-5.7716990462030536E-18,-4.7925971188595567E-17,
        5.9360068943581368E-18,-6.1272563459363171E-17,5.0279875749015268E-18,-0.2270746709188694,
        -1.1826274009564541E-17,8.3068944653702861E-17,-3.8692465030576439E-18,-0.22709222314756114,
        -5.7716990462030536E-18,-4.7925971188595567E-17,-9.1547320939244781E-18,-0.22709254163278178,
        -0.024691844478350409,7.8430168718064686E-17,-0.024691844478350409,2.5117660907994846E-16,
        -4.7238965429826388E-18,1.0376068900570454E-16,-0.024695431618763558,2.0548256970736797E-16,
        -1.5720931501039814E-17,-6.1264569585923459E-17,-0.024688864080425831,-8.9425503406372758E-17,
        1.7767363101606204E-17,-0.22709222314756114,1.5666721392415539E-17,-0.22707467091886915,
        1.0164395367051604E-17,-0.40515003408376971,-7.1692868655603981E-18,-2.8378144831860824E-17,
        -5.7716990462030536E-18,-4.7925971188595567E-17,5.082197683525802E-18,-0.22707467091886949,
        -1.463672932855431E-17,-0.22709222314756122,-0.024694734132731256,1.6721192708452418E-16,
        -0.040652897782438434,2.1352006534386403E-17,-0.024682330526772954,-0.22709121837416038,
        1.1786722988960778E-18,-1.8853815205357853E-16,-1.7381116077658243E-18,-2.3392575078771017E-17,
        1.10285525039494E-18,1.5792918713644589E-16,-4.7470079692973704E-18,-6.9875982983743506E-17,
        -4.645797251472679E-18,-6.9338328820473839E-17,1.148179112794923E-18,-1.8854191076228197E-16,
        -1.0777346329819693E-17,8.4682682732228818E-20,0.90852126123084109,0.043908146081154252,
        -1.1237416704633352E-16,0.044340059223466725,0.90854213589311628,-5.4210108624275222E-18,
        0.22499743169378195,0.044391150716473024,0.90854320277576739,0.013973130057841329,0.40175302414947389,
        0.044302834795567785,0.90853861186181406,0.02289738328452481,-1.1237416704633352E-16,0.044340059223466725,
        0.90854213589311628,-5.4210108624275222E-18,0.22499743169378195,0.044391150716473024,0.90854320277576739,
        0.013973130057841329,0.40175302414947389,0.044302834795567785,0.90853861186181406,0.02289738328452481,
        2.0211137857729586E-16,3.3610267347050637E-18,-1.4233541645661263E-17,0.044446387153773116,
        1.2255042087464668E-16,0.014073066200566241,1.7068052700353054E-16,0.044433312973263257,
        1.4178653910679184E-16,0.02308043023166,2.0211137857729586E-16,3.3610267347050637E-18,
        1.2254660922638404E-16,0.014073066200566246,1.4178653910679184E-16,0.02308043023166,0.22500289657472694,
        -1.6127507315721878E-18,0.90854626790451765,-5.4210108624275222E-19,0.4017626395980568,
        -1.0543866127421531E-17,0.90854551524313676,-7.48099499014998E-18,2.9203154922486513E-17,
        -7.37257477290143E-18,0.22500289657472694,-1.6127507315721878E-18,0.40176263959805669,
        -1.0489656018797255E-17,0.2250031571391346,0.014084282907403574,0.22500194445913865,0.023101232532859166,
        0.22500289657472694,-1.7821573210230479E-17,0.2250031571391346,0.014084282907403586,0.40176311984350016,
        0.014063877541696803,1.2255465603938295E-16,0.014073066200566236,0.2250031571391346,0.014084282907403574,
        0.40176311984350005,0.014063877541696803,0.4017609942320583,0.023063772260979193,0.40176263959805669,
        -5.0957502106818708E-18,0.40176311984350022,0.014063877541696813,0.4017609942320583,0.023063772260979193,
        -2.0403837853229939E-16,0.02308043023166,0.22500194445913849,0.023101232532859169,0.401760994232058,
        0.023063772260979186,2.0211137857729586E-16,3.3610267347050637E-18,-1.4233541645661263E-17,
        0.044446387153773116,1.2254660922638404E-16,0.014073066200566246,-1.9888333601530972E-18,
        0.044433312973263257,1.4178653910679184E-16,0.02308043023166,0.22500289657472694,-1.6127507315721878E-18,
        0.90854626790451765,-5.9631119486702744E-18,0.40176263959805669,-1.0489656018797255E-17,0.90854551524313676,
        -7.48099499014998E-18,0.2250031571391346,0.014084282907403586,0.22500194445913865,0.023101232532859166,
        0.40176311984350005,0.014063877541696808,0.40176099423205819,0.023063772260979193,1.1948500863853337E-16,
        7.8316666303132609E-18,1.0077230382823216E-16,2.5478751053409354E-18,4.0905762121751926E-17,
        -1.6703489719854803E-18,8.65074749030817E-18,0.014073452133259199,5.3407121390278145E-17,
        0.023119416718676764,1.0077092739969287E-16,2.5343225781848666E-18,8.643971226730135E-18,
        0.014073452133259209,0.22502056771591866,-8.2263839837337649E-18,0.40176453880416918,
        -6.5323180892251642E-18,0.90854657053851451,-5.5294310796760726E-18,-2.45051555019675E-16,
        -2.6834003769016235E-18,0.22500396954755839,-9.4867690092481638E-19,0.40176453880416907,
        -6.478107980600889E-18,0.40176467697335466,2.439454888092385E-19,-5.3732382042023796E-17,
        -8.3331101350878067E-18,4.1341984089587891E-17,-7.0235971986326584E-18,0.22502056771591855,
        -8.1518450843753865E-18,0.22501961554900995,0.023105898263657981,0.22500396954755847,
        -1.1858461261560205E-17,0.225003234379625,0.014084670139843564,5.3978445113201171E-17,0.014094294168846267,
        0.22502082855573682,0.014086833295573026,0.40176453880416929,-6.6407383064737147E-18,0.40176418862008356,
        -6.3967928176644762E-18,0.40176325784096573,0.014064262811759857,-1.1939607017907167E-16,
        0.023119416718676764,0.22501961554900987,0.023105898263657981,4.1339442990746128E-17,
        -1.6195269951502222E-18,4.3272795692854069E-18,-2.1819568721270777E-18,8.3520836731063031E-17,
        0.023124920378727248,5.4079242033924432E-17,0.014094294168846278,8.643971226730135E-18,0.014073452133259209,
        2.2653726767726812E-16,0.023119416718676764,0.22502056771591855,-8.1518450843753865E-18,0.22500376942411082,
        -4.2283884726934673E-18,0.90854657053851451,-1.0950441942103595E-17,0.225020828555737,0.014086833295573026,
        0.225003234379625,0.014084670139843564,0.4017632578409655,0.014064262811759858,6.8140584528386856E-17,
        4.7298319774680131E-18,1.5717712775840248E-16,4.8427867988345792E-18,1.8241786255363338E-16,
        0.014099813725742058,9.7153620258884181E-18,-1.44774871344705E-17,1.9124479289697044E-16,
        0.014094682296279696,6.8139128690508763E-17,4.7162794503119443E-18,6.6146920433456449E-17,
        0.014097649905087963,0.22502164116342194,-6.8711312681268844E-18,0.2250216411634221,-1.5517643593698782E-18,
        1.0201159574812646E-16,-2.2158381900172497E-18,0.22502171855946634,-2.1480755542369057E-18,
        -1.5798011499239956E-17,-4.91865166871488E-19,0.22502144099999252,-2.6766241133235891E-18,
        1.8120999357084874E-17,0.014094682296279686,9.6193296654934618E-18,0.014099813725742047,
        -1.9217822320484468E-16,0.023129589494450122,1.5185585502551415E-16,3.1611269591530489E-18,
        6.8139128690508763E-17,4.7162794503119443E-18,9.698950762535366E-18,0.014099813725742063,
        1.9135406014716624E-16,0.014094682296279696,0.22500404688447739,-8.40256683676266E-18,0.40176467697335472,
        -1.0625181290357943E-17,0.22502090585531667,0.0140872207964491,2.8013481348918148E-16,
        -5.2482161411876449E-18,1.0580415599095554E-16,2.786738913454531E-18,1.0705883760614638E-16,
        -1.0608240631412857E-17,1.0176638301861879E-16,-2.2463313761184045E-18,1.0165657313794115E-16,
        3.1509625637859973E-18,2.8013342961601668E-16,-5.2583805365546965E-18,5.7474348667278365E-20,
        2.9607205860406696E-20,0.077953938048960669,0.91495630205656719,-1.5395670849294163E-17,0.91499336154188149,
        0.078388923478923359,1.2000762796698927E-17,0.024548090137893282,0.91499404071464974,0.0784581439271197,
        0.22706440144138565,0.040393877243513461,0.91498555513722191,0.07837495020825766,0.405131234178429,
        -1.5395670849294163E-17,0.91499336154188149,0.078388923478923359,1.2000762796698927E-17,
        0.024548090137893282,0.91499404071464974,0.0784581439271197,0.22706440144138565,0.040393877243513461,
        0.91498555513722191,0.07837495020825766,0.405131234178429,1.2197274440461925E-18,6.8118389618190833E-17,
        4.9873299934333204E-18,0.91500006722362592,4.8382521947165635E-18,0.22707303152550876,
        3.2526065174565133E-18,0.91499867394199985,9.7849246066816775E-18,0.4051470246964986,1.2197274440461925E-18,
        6.8118389618190833E-17,4.8382521947165635E-18,0.22707303152550876,9.7849246066816775E-18,0.4051470246964986,
        0.024660732712307117,-1.417594340524797E-17,0.078507952497007219,-1.9447876468958736E-17,
        0.040592464909515784,-1.8488357546309064E-16,0.078497094095205028,-7.5948362182609586E-17,
        1.3823577699190182E-18,-2.7769805769142786E-16,0.024660732712307103,-1.4168320108722682E-17,
        0.040592464909515784,-1.8488357546309064E-16,0.024678049245177087,0.22707314681162666,0.02465616095779212,
        0.405147254584257,0.024660732712307117,-1.8708416706005732E-16,0.024678049245177087,0.22707314681162666,
        0.0406235469714099,0.22707117636130061,-5.9089018400459992E-18,0.22707303152550867,0.024678049245177074,
        0.22707314681162657,0.0406235469714099,0.22707117636130061,0.040585198407018679,0.405143641589301,
        0.040592464909515784,-1.1975351808281298E-17,0.040623546971409907,0.2270711763613007,0.040585198407018679,
        0.405143641589301,-1.1763593571467723E-17,0.40514702469649849,0.0246561609577921,0.405147254584257,
        0.040585198407018672,0.405143641589301,1.2197274440461925E-18,6.8118389618190833E-17,4.9873299934333204E-18,
        0.91500006722362592,4.8382521947165635E-18,0.22707303152550876,3.2526065174565133E-18,0.91499867394199985,
        9.7849246066816775E-18,0.4051470246964986,0.024660732712307103,-1.4168320108722682E-17,0.078507952497007219,
        -1.9447876468958736E-17,0.040592464909515784,-1.8488357546309064E-16,0.078497094095205028,
        -7.5948362182609586E-17,0.024678049245177087,0.22707314681162666,0.024656160957792109,0.405147254584257,
        0.0406235469714099,0.22707117636130061,0.040585198407018679,0.405143641589301,1.4094628242311558E-18,
        -6.5815518792843204E-18,1.4894227344519617E-17,4.6953577365147631E-17,-7.3183646642771549E-19,
        1.4633468251707381E-16,-5.2922618544448685E-18,0.22709100233229687,9.5680841721845766E-18,
        0.40514926269585039,1.4894227344519617E-17,4.6953577365147631E-17,-5.2922618544448685E-18,
        0.22709100233229687,0.02466142784965503,-1.1036924006018259E-16,0.040646457087583146,
        -1.5888644024596166E-17,0.0785223958657716,-8.3937576941112146E-17,-2.8192644616412132E-17,
        -2.9900517147960978E-16,0.02469114725936063,-9.6381337969225073E-17,0.040646457087583146,
        -1.5888644024596166E-17,0.040652897782438434,-1.9426361832098477E-16,1.5178830414797062E-18,
        -1.7948585800671261E-16,-6.5052130349130266E-19,-2.657311762126191E-17,0.02466142784965503,
        -1.1037008709312984E-16,0.024656855942051376,0.40514743808224646,0.024691147259360651,
        -9.639658456227565E-17,0.024681633887332338,0.22709111782296573,-7.15573433840433E-18,0.22707425188322058,
        0.024678745617735788,0.22707324731405812,0.040646457087583153,-1.5893726222279692E-17,0.040641311777483369,
        -4.953956895311501E-17,0.04062998370810441,0.22708914685042259,-1.0299920638612292E-18,0.40514926269585017,
        0.024656855942051355,0.40514743808224646,-7.3183646642771549E-19,1.4633468251707381E-16,
        2.0464316005663896E-18,2.880081427254072E-17,-6.2341624917916505E-18,0.40514985034555978,
        -7.26415455565288E-18,0.22707425188322075,-5.2922618544448685E-18,0.22709100233229687,
        9.5680841721845766E-18,0.40514926269585039,0.02466142784965503,-1.1037008709312984E-16,0.02468816702271235,
        -1.2348385118252092E-16,0.0785223958657716,-8.3937576941112146E-17,0.0246787456177358,0.22707324731405804,
        0.024681633887332327,0.22709111782296573,0.040629983708104396,0.22708914685042267,5.7716990462030536E-18,
        4.7925971188595567E-17,-5.9360068943581368E-18,6.1272563459363171E-17,-5.0279875749015268E-18,
        0.2270746709188694,1.1826274009564541E-17,-8.3068944653702861E-17,3.8692465030576439E-18,
        0.22709222314756114,5.7716990462030536E-18,4.7925971188595567E-17,9.1547320939244781E-18,
        0.22709254163278178,0.024691844478350409,-7.8430168718064686E-17,0.024691844478350409,
        -2.5117660907994846E-16,4.7238965429826388E-18,-1.0376068900570454E-16,0.024695431618763558,
        -2.0548256970736797E-16,1.5720931501039814E-17,6.1264569585923459E-17,0.024688864080425831,
        8.9425503406372758E-17,-1.7767363101606204E-17,0.22709222314756114,-1.5666721392415539E-17,
        0.22707467091886915,-1.0164395367051604E-17,0.40515003408376971,7.1692868655603981E-18,
        2.8378144831860824E-17,5.7716990462030536E-18,4.7925971188595567E-17,-5.082197683525802E-18,
        0.22707467091886949,1.463672932855431E-17,0.22709222314756122,0.024694734132731256,-1.6721192708452418E-16,
        0.040652897782438434,-2.1352006534386403E-17,0.024682330526772954,0.22709121837416038,
        -1.1786722988960778E-18,1.8853815205357853E-16,1.7381116077658243E-18,2.3392575078771017E-17,
        -1.10285525039494E-18,-1.5792918713644589E-16,4.7470079692973704E-18,6.9875982983743506E-17,
        4.645797251472679E-18,6.9338328820473839E-17,-1.148179112794923E-18,1.8854191076228197E-16,
        1.0777346329819693E-17,-8.4682682732228818E-20,-0.0032231717786674243,-0.00047387004623103532,-1.0,
        1.0842021724855044E-19,-0.0032233970643617714,1.5670109524204556E-20,-0.50017152346648186,
        -0.00012270693090584496,-0.003223438748220626,-0.0001096414616121335,-0.33389281505076362,
        -0.00021633303651176036,-0.0032233972588470859,-0.00020082461188265349,-1.0,1.0842021724855044E-19,
        -0.0032233970643617714,1.5670109524204556E-20,-0.50017152346648186,-0.00012270693090584496,
        -0.003223438748220626,-0.00010964146161213346,-0.33389281505076362,-0.00021633303651176036,
        -0.0032233972588470859,-0.00020082461188265349,-1.0,5.4210108624275222E-20,-1.0,0.0,-1.0,
        -1.0842021724855044E-19,-1.0,0.0,-1.0,0.0,-1.0,5.4210108624275222E-20,-1.0,0.0,-1.0,0.0,-0.500171538572618,
        0.0,-0.0032234627990377889,3.7692966152816365E-20,-0.33389286200349694,5.4210108624275222E-20,
        -0.0032234578058911562,6.5645053412208276E-20,-0.99999999999999978,5.4210108624275222E-20,
        -0.500171538572618,0.0,-0.33389286200349694,5.4210108624275222E-20,-0.50017154120112894,
        -2.8830983828423548E-5,-0.50017153832237338,-5.2621143293484158E-5,-0.500171538572618,0.0,
        -0.50017154120112894,-2.8830983828423494E-5,-0.33389287043993776,-5.0429547165299263E-5,-1.0,0.0,
        -0.50017154120112894,-2.8830983828423548E-5,-0.33389287043993776,-5.0429547165299263E-5,-0.3338928616111102,
        -9.2256767123402269E-5,-0.333892862003497,2.7105054312137611E-20,-0.33389287043993771,
        -5.0429547165299263E-5,-0.3338928616111102,-9.2256767123402269E-5,-1.0000000000000002,
        5.4210108624275222E-20,-0.50017153832237338,-5.2621143293484266E-5,-0.33389286161111031,
        -9.225676712340216E-5,-1.0,5.4210108624275222E-20,-1.0,0.0,-1.0,0.0,-1.0,0.0,-1.0,0.0,-0.500171538572618,
        0.0,-0.0032234627990377889,3.7269449679189215E-20,-0.33389286200349694,5.4210108624275222E-20,
        -0.0032234578058911562,6.5645053412208276E-20,-0.50017154120112894,-2.8830983828423494E-5,
        -0.50017153832237338,-5.2621143293484158E-5,-0.33389287043993776,-5.0429547165299263E-5,-0.3338928616111102,
        -9.2256767123402269E-5,-1.0,5.4210108624275222E-20,-1.0,5.4210108624275222E-20,-1.0,5.4210108624275222E-20,
        -1.0,0.0,-1.0,0.0,-1.0,5.4210108624275222E-20,-1.0,5.4210108624275222E-20,-0.50017155139325642,
        5.4210108624275222E-20,-0.33389287552797581,0.0,-0.0032234713063484617,3.7269449679189215E-20,-1.0,
        1.6263032587282567E-19,-0.50017154286415544,0.0,-0.33389287552797581,0.0,-0.3338928772195392,
        5.4210108624275222E-20,-1.0,1.0842021724855044E-19,-0.99999999999999978,1.0842021724855044E-19,
        -0.50017155139325642,5.4210108624275222E-20,-0.50017155114301959,-5.2624528352597055E-5,
        -0.50017154286415533,-5.4210108624275222E-20,-0.50017154172544676,-2.8833612408983415E-5,-1.0,0.0,
        -0.50017155402213676,-2.8832834192057944E-5,-0.3338928755279757,-2.7105054312137611E-20,
        -0.33389287438889476,8.1315162936412833E-20,-0.33389287213054836,-5.0434267119571795E-5,-1.0000000000000002,
        1.6263032587282567E-19,-0.50017155114301959,-5.2624528352597164E-5,-1.0,5.4210108624275222E-20,-1.0,
        5.4210108624275222E-20,-1.0,0.0,-1.0,5.4210108624275222E-20,-1.0,5.4210108624275222E-20,-1.0,0.0,
        -0.50017155139325642,5.4210108624275222E-20,-0.5001715424793699,-5.4210108624275222E-20,
        -0.0032234713063484617,3.7269449679189215E-20,-0.50017155402213676,-2.8832834192057835E-5,
        -0.50017154172544676,-2.8833612408983415E-5,-0.33389287213054852,-5.0434267119571713E-5,-1.0,
        5.4210108624275222E-20,-0.99999999999999978,0.0,-0.99999999999999978,-5.4210108624275222E-20,-1.0,
        5.4210108624275222E-20,-1.0,5.4210108624275222E-20,-1.0,5.4210108624275222E-20,-1.0,0.0,
        -0.50017155568537663,5.4210108624275222E-20,-0.50017155568537675,0.0,-1.0,5.4210108624275222E-20,
        -0.50017155621007536,0.0,-1.0,1.6263032587282567E-19,-0.50017155530055091,0.0,-1.0,-5.4210108624275222E-20,
        -0.99999999999999978,-1.6263032587282567E-19,-1.0,5.4210108624275222E-20,-1.0,5.4210108624275222E-20,-1.0,
        5.4210108624275222E-20,-0.99999999999999978,-5.4210108624275222E-20,-1.0,5.4210108624275222E-20,
        -0.50017154338877634,0.0,-0.3338928772195392,2.7105054312137611E-20,-0.500171554546532,
        -2.883546297236672E-5,-1.0,5.4210108624275222E-20,-0.99999999999999978,0.0,-1.0,5.4210108624275222E-20,-1.0,
        5.4210108624275222E-20,-1.0,5.4210108624275222E-20,-1.0,5.4210108624275222E-20,-0.99999999999999978,0.0,
        -0.00047387004623103553,-0.0032530855295321241,-4.1504614415460717E-20,-0.00325331080846554,
        -5.4210108624275222E-20,-0.99999999999999989,-0.00012270693090584504,-0.003253333675105293,
        -0.0001096414616121335,-0.50017290377260126,-0.00021633303651176052,-0.0032532861083053037,
        -0.00020082461188265359,-0.33389770950648251,-4.1504614415460717E-20,-0.00325331080846554,
        -5.4210108624275222E-20,-0.99999999999999989,-0.00012270693090584504,-0.003253333675105293,
        -0.0001096414616121335,-0.50017290377260126,-0.00021633303651176052,-0.0032532861083053037,
        -0.00020082461188265359,-0.33389770950648251,0.0,-0.99999999999999989,-1.300195574035351E-19,
        -0.0032533637994211317,-5.4210108624275222E-20,-0.50017291583272638,-1.0418505251227894E-19,
        -0.0032533563672422191,-5.4210108624275222E-20,-0.33389774996742894,0.0,-0.99999999999999989,
        -5.4210108624275222E-20,-0.50017291583272638,-5.4210108624275222E-20,-0.33389774996742894,
        -1.0842021724855044E-19,-0.99999999999999989,0.0,-1.0,-1.0842021724855044E-19,-0.99999999999999989,
        -5.4210108624275222E-20,-0.99999999999999989,-1.0842021724855044E-19,-0.99999999999999989,
        -1.0842021724855044E-19,-0.99999999999999989,-1.0842021724855044E-19,-0.99999999999999989,
        -2.8830983828423494E-5,-0.500172916913477,-5.2621143293484266E-5,-0.3338977537047928,0.0,-1.0,
        -2.8830983828423494E-5,-0.500172916913477,-5.0429547165299344E-5,-0.50017291437548894,
        -5.4210108624275222E-20,-0.50017291583272638,-2.8830983828423385E-5,-0.50017291691347721,
        -5.0429547165299344E-5,-0.50017291437548894,-9.2256767123402269E-5,-0.33389774515228049,
        -1.0842021724855044E-19,-0.99999999999999989,-5.0429547165299344E-5,-0.50017291437548894,
        -9.2256767123402269E-5,-0.33389774515228049,1.0842021724855044E-19,-0.333897749967429,
        -5.2621143293484212E-5,-0.3338977537047928,-9.2256767123402215E-5,-0.33389774515228055,0.0,
        -0.99999999999999989,-1.300195574035351E-19,-0.0032533637994211317,-5.4210108624275222E-20,
        -0.50017291583272638,-1.0418505251227894E-19,-0.0032533563672422191,-5.4210108624275222E-20,
        -0.33389774996742894,-1.0842021724855044E-19,-0.99999999999999989,0.0,-1.0,-1.0842021724855044E-19,
        -0.99999999999999989,-5.4210108624275222E-20,-0.99999999999999989,-2.8830983828423494E-5,-0.500172916913477,
        -5.2621143293484266E-5,-0.3338977537047928,-5.0429547165299344E-5,-0.50017291437548894,
        -9.2256767123402269E-5,-0.33389774515228049,0.0,-0.99999999999999989,0.0,-0.99999999999999989,
        -1.0842021724855044E-19,-0.99999999999999989,-5.4210108624275222E-20,-0.50017292901042176,
        -1.0842021724855044E-19,-0.33389775792997123,0.0,-0.99999999999999989,-5.4210108624275222E-20,
        -0.50017292901042176,-1.0842021724855044E-19,-0.99999999999999989,-1.0842021724855044E-19,
        -0.99999999999999989,-5.4210108624275222E-20,-0.99999999999999989,-5.4210108624275222E-20,
        -0.99999999999999989,-1.0842021724855044E-19,-0.99999999999999989,-1.0842021724855044E-19,
        -0.99999999999999989,-1.0842021724855044E-19,-0.99999999999999989,-5.4210108624275222E-20,
        -0.99999999999999989,-5.4210108624275222E-20,-0.99999999999999989,-1.0842021724855044E-19,
        -0.99999999999999989,-5.2624528352597055E-5,-0.33389775459855631,0.0,-1.0,-2.8833612408983415E-5,
        -0.50017293009143149,-5.4210108624275222E-20,-0.50017291819340215,-2.8832834192057727E-5,
        -0.50017291718052692,-1.0842021724855044E-19,-0.99999999999999989,-5.4210108624275222E-20,
        -0.99999999999999989,-5.0434267119571822E-5,-0.50017292755295606,5.4210108624275222E-20,
        -0.33389775792997128,-5.2624528352597055E-5,-0.33389775459855625,-1.0842021724855044E-19,
        -0.99999999999999989,0.0,-0.99999999999999989,-5.4210108624275222E-20,-0.33389775924466275,0.0,
        -0.500172918193402,-5.4210108624275222E-20,-0.50017292901042176,-1.0842021724855044E-19,
        -0.33389775792997123,-1.0842021724855044E-19,-0.99999999999999989,-5.4210108624275222E-20,
        -0.99999999999999989,-5.4210108624275222E-20,-0.99999999999999989,-2.8832834192057781E-5,
        -0.5001729171805267,-2.8833612408983415E-5,-0.50017293009143149,-5.0434267119571822E-5,-0.50017292755295606,
        0.0,-0.99999999999999989,-5.4210108624275222E-20,-0.99999999999999989,5.4210108624275222E-20,
        -0.50017291884376192,-1.0842021724855044E-19,-0.99999999999999989,0.0,-0.50017293137158414,0.0,
        -0.99999999999999989,-5.4210108624275222E-20,-0.50017293175475663,-1.0842021724855044E-19,
        -0.99999999999999989,-1.0842021724855044E-19,-0.99999999999999989,-5.4210108624275222E-20,
        -0.99999999999999989,-1.0842021724855044E-19,-0.99999999999999989,-5.4210108624275222E-20,
        -0.99999999999999989,-1.0842021724855044E-19,-0.99999999999999989,-1.6263032587282567E-19,
        -0.500172931371584,0.0,-0.50017291884376214,5.4210108624275222E-20,-0.33389776013913919,
        -1.0842021724855044E-19,-0.99999999999999989,0.0,-0.99999999999999989,5.4210108624275222E-20,
        -0.50017291884376192,0.0,-0.50017293137158414,-1.0842021724855044E-19,-0.99999999999999989,
        -1.0842021724855044E-19,-0.99999999999999989,-2.8835462972366666E-5,-0.50017293035853716,0.0,
        -0.99999999999999989,-5.4210108624275222E-20,-0.99999999999999989,-1.0842021724855044E-19,
        -0.99999999999999989,-1.6263032587282567E-19,-0.99999999999999989,0.0,-0.99999999999999989,0.0,
        -0.99999999999999989,0.0,-0.99999999999999989];
END_VAR

VAR_TEMP
    new_x: ARRAY [0..5] OF LREAL;
    y_innov: ARRAY [0..1] OF LREAL;
    th: ARRAY [0..9] OF LREAL;
    b_k: DINT;
    du: ARRAY [0..1] OF LREAL;
    found: BOOL;
    regionmin: DINT;
    betamin: LREAL;
    beta: LREAL;
    betah: LREAL;
    b_h: DINT;
    rtb_xest: ARRAY [0..5] OF LREAL;
    i: DINT;
    rtb_last_mv_idx_0: LREAL;
    rtb_last_mv_idx_1: LREAL;
END_VAR

CASE ssMethodType OF
    SS_INITIALIZE: 
        (* SystemInitialize for Atomic SubSystem: '<Root>/Explicit Controller' *)
        (* InitializeConditions for Memory: '<S3>/last_x' *)
        FOR i := 0 TO 5 DO 
            last_x_PreviousInput[i] := 0.0;
        END_FOR;
        (* End of InitializeConditions for Memory: '<S3>/last_x' *)
        
        (* InitializeConditions for UnitDelay: '<S3>/last_mv' *)
        last_mv_DSTATE[0] := 0.0;
        last_mv_DSTATE[1] := 0.0;
        (* End of SystemInitialize for SubSystem: '<Root>/Explicit Controller' *)
    SS_STEP: 
        (* Outputs for Atomic SubSystem: '<Root>/Explicit Controller' *)
        (* MATLAB Function: '<S3>/Explicit MPC Evaluation' *)
        (* MATLAB Function 'Explicit MPC Controller/MPC/Explicit MPC Evaluation': '<S4>:1' *)
        (* '<S4>:1:6' coder.extrinsic('mpcblock_pwa_evaluate_double_mex'); *)
        (* '<S4>:1:7' coder.extrinsic('mpcblock_pwa_evaluate_single_mex'); *)
        (* Parameters *)
        (* '<S4>:1:10' isSimulation = coder.target('Sfun') && ~coder.target('RtwForRapid') && ~coder.target('RtwForSim'); *)
        (* '<S4>:1:11' isDouble = isa(r,'double'); *)
        (* '<S4>:1:12' ZERO = zeros('like',r); *)
        (* '<S4>:1:13' ONE = ones('like',r); *)
        (* Pre-allocate all the MEX block outputs for the simulation mode *)
        (* '<S4>:1:18' if isSimulation *)
        (* '<S4>:1:26' if isSimulation *)
        (* '<S4>:1:39' else *)
        (* When doing code generation, use M code directly *)
        (* '<S4>:1:41' [u, status, region, new_x, xest] = mpcblock_pwa_evaluate(old_x, r, v, ym, ext_u, old_u, no_mv, nu, nx, nv, uoff, ... *)
        (* '<S4>:1:42'         openloopflag, F, G, H, K, i1, i2, nr, np, xunfindex, refunfindex, uunfindex, mdunfindex,thmin,thmax,... *)
        (* '<S4>:1:43'         CustomEstimation, RMYscale, myoff, xoff, A, Bu, Bv, Cm, Dvm, M, L, ... *)
        (* '<S4>:1:44'         switch_in, switch_inport, no_switch, enable_value); *)
        regionmin := 1;
        b_k := -1;
        (* End of Outputs for SubSystem: '<Root>/Explicit Controller' *)
        (* Outputs for Atomic SubSystem: '<Root>/Explicit Controller' *)
        (* MATLAB Function: '<S3>/Explicit MPC Evaluation' incorporates:
         *  Memory: '<S3>/last_x' *)
        FOR i := 0 TO 5 DO 
            new_x[i] := last_x_PreviousInput[i];
        END_FOR;
        (* End of Outputs for SubSystem: '<Root>/Explicit Controller' *)
        (* Outputs for Atomic SubSystem: '<Root>/Explicit Controller' *)
        (* MATLAB Function: '<S3>/Explicit MPC Evaluation' *)
        FOR i := 0 TO 1 DO 
            betamin := 0.0;
            FOR b_h := 0 TO 5 DO 
                betamin := (Explicit_b_Cm[(b_h * 2) + i] * new_x[b_h]) + betamin;
            END_FOR;
            y_innov[i] := MeasuredTankOutputs[i] - betamin;
        END_FOR;
        (* End of Outputs for SubSystem: '<Root>/Explicit Controller' *)
        (* Outputs for Atomic SubSystem: '<Root>/Explicit Controller' *)
        (* MATLAB Function: '<S3>/Explicit MPC Evaluation' *)
        FOR i := 0 TO 5 DO 
            rtb_xest[i] := ((Explicit_b_M[i + 6] * y_innov[1]) + (Explicit_b_M[i] * y_innov[0])) + new_x[i];
        END_FOR;
        (* End of Outputs for SubSystem: '<Root>/Explicit Controller' *)
        (* Outputs for Atomic SubSystem: '<Root>/Explicit Controller' *)
        (* MATLAB Function: '<S3>/Explicit MPC Evaluation' incorporates:
         *  UnitDelay: '<S3>/last_mv' *)
        FOR i := 0 TO 9 DO 
            th[i] := 0.0;
        END_FOR;
        FOR b_h := 0 TO 5 DO 
            th[b_h] := rtb_xest[b_h];
        END_FOR;
        th[6] := ref[0];
        th[8] := last_mv_DSTATE[0];
        th[7] := ref[1];
        th[9] := last_mv_DSTATE[1];
        FOR b_h := 0 TO 9 DO 
            betamin := th[b_h];
            IF betamin < Explicit_b_thmin[b_h] THEN 
                regionmin := 0;
            ELSIF betamin > Explicit_b_thmax[b_h] THEN 
                regionmin := 0;
            END_IF;
        END_FOR;
        du[0] := 0.0;
        du[1] := 0.0;
        IF regionmin = 1 THEN 
            found := FALSE;
            regionmin := 0;
            betamin := 1.797693134862316E+307;
            WHILE ( NOT found) AND ((b_k + 1) < 125) DO
                b_k := b_k + 1;
                b_h := INT_TO_DINT(b_i1[b_k]);
                beta := -1.0;
                WHILE b_h <= INT_TO_DINT(b_i2[b_k]) DO
                    betah := 0.0;
                    FOR i := 0 TO 9 DO 
                        betah := (Explicit_g_H[((2526 * i) + b_h) - 1] * th[i]) + betah;
                    END_FOR;
                    betah := betah - Explicit_c_K[b_h - 1];
                    IF betah > beta THEN 
                        beta := betah;
                    END_IF;
                    b_h := b_h + 1;
                END_WHILE;
                IF beta <= 0.0 THEN 
                    found := TRUE;
                ELSIF betamin > beta THEN 
                    betamin := beta;
                    regionmin := b_k + 1;
                END_IF;
            END_WHILE;
            IF  NOT found THEN 
                b_k := regionmin - 1;
            END_IF;
            b_k := DWORD_TO_DINT(SHL(DINT_TO_DWORD(b_k), 1));
            FOR regionmin := 0 TO 1 DO 
                b_h := regionmin + b_k;
                betamin := 0.0;
                FOR i := 0 TO 9 DO 
                    betamin := (Explicit_b_F[(250 * i) + b_h] * th[i]) + betamin;
                END_FOR;
                du[regionmin] := Explicit_b_G[regionmin + b_k] + betamin;
            END_FOR;
        END_IF;
        betamin := last_mv_DSTATE[0] + du[0];
        beta := betamin;
        mv[0] := betamin;
        betamin := last_mv_DSTATE[1] + du[1];
        (* End of Outputs for SubSystem: '<Root>/Explicit Controller' *)
        (* Outputs for Atomic SubSystem: '<Root>/Explicit Controller' *)
        FOR i := 0 TO 5 DO 
            (* MATLAB Function: '<S3>/Explicit MPC Evaluation' *)
            rtb_xest[i] := 0.0;
            FOR b_h := 0 TO 5 DO 
                rtb_xest[i] := (Explicit_b_A[(6 * b_h) + i] * new_x[b_h]) + rtb_xest[i];
            END_FOR;
            (* Update for Memory: '<S3>/last_x' incorporates:
             *  MATLAB Function: '<S3>/Explicit MPC Evaluation' *)
            last_x_PreviousInput[i] := ((Explicit_b_L[i + 6] * y_innov[1]) + (Explicit_b_L[i] * y_innov[0])) + (rtb_xest[i] + ((Explicit_b_Bu[i + 6] * betamin) + (Explicit_b_Bu[i] * beta)));
        END_FOR;
        (* Update for UnitDelay: '<S3>/last_mv' *)
        last_mv_DSTATE[0] := mv[0];
        (* Outport: '<Root>/mv' incorporates:
         *  Gain: '<S3>/ext.mv_scale1'
         *  UnitDelay: '<S3>/last_mv' *)
        mv[0] := 0.15299877600979192 * mv[0];
        (* Update for UnitDelay: '<S3>/last_mv' *)
        last_mv_DSTATE[1] := betamin;
        (* Outport: '<Root>/mv' incorporates:
         *  Gain: '<S3>/ext.mv_scale1' *)
        mv[1] := 0.15299877600979192 * betamin;
        (* End of Outputs for SubSystem: '<Root>/Explicit Controller' *)
END_CASE;

IF FOUND THEN
	search_status := TRUE;
ELSE 
	search_status := FALSE;
END_IF

END_FUNCTION_BLOCK
